PROGRAM Drain
VAR
	nSource: INT;
	nStartTimeInSeconds: UDINT ;
	nTime: UDINT;
	tempSecondsToAddWhilePause: INT;
	SecondsToAddWhilePause: INT;
	RemainingTime: UDINT;
	fb_FTRIG: R_TRIG;
	bStartCommand: BOOL;
	CLK: INT;
	Q: INT;
	b: BOOL;
	bN2PurgeBlockEnded: BOOL;
	fbSelection : FBSelection;
	

END_VAR

VAR_INPUT
	nCurrentBlock: INT;
	sSourceName: STRING;
END_VAR

fbSelection.TargetConverter(sTargetName:= sSourceName, TargetConverter_output => nSource); 


IF (RecipeTags.bStartTimeEnable[nCurrentBlock]=FALSE) THEN
	RecipeTags.Recipe.Blocks[nCurrentBlock].Properties.sStartTime:=MAIN.sConcatenatedHourMinuteString;
	nStartTimeInSeconds := STRING_TO_UDINT(MAIN.sCurrentSecond);
	RecipeTags.bStartTimeEnable[nCurrentBlock] :=  TRUE;
END_IF



IF RecipeTags.Recipe.Blocks[nCurrentBlock].Properties.sIntervalType = 'S' THEN
	nTime := DINT_TO_UDINT(RecipeTags.Recipe.Blocks[nCurrentBlock].Properties.nInterval);
ELSIF RecipeTags.Recipe.Blocks[nCurrentBlock].Properties.sIntervalType = 'M' THEN
	nTime := DINT_TO_UDINT(RecipeTags.Recipe.Blocks[nCurrentBlock].Properties.nInterval * 60);
ELSIF RecipeTags.Recipe.Blocks[nCurrentBlock].Properties.sIntervalType = 'H' THEN
	nTime := DINT_TO_UDINT(RecipeTags.Recipe.Blocks[nCurrentBlock].Properties.nInterval * 3600);
END_IF


IF RecipeTags.enWaitPause[nCurrentBlock] THEN
	tempSecondsToAddWhilePause := tempSecondsToAddWhilePause + 1;
	SecondsToAddWhilePause := tempSecondsToAddWhilePause; 
ELSE
	tempSecondsToAddWhilePause := 0;
END_IF

IF NOT(RecipeTags.bPauseRecipe) THEN
		RecipeTags.enWaitPause[nCurrentBlock] := FALSE;
		RecipeTags.bBlockStart[nCurrentBlock] := TRUE;
		RemainingTime := nTime- nStartTimeInSeconds-STRING_TO_UDINT(MAIN.sCurrentSecond);
ELSE
		RecipeTags.bBlockStart[nCurrentBlock] := FALSE;
		RecipeTags.enWaitPause[nCurrentBlock] := TRUE;
END_IF

IF  (nTime + nStartTimeInSeconds + DINT_TO_UDINT(TRUNC(SecondsToAddWhilePause/100))) <= (STRING_TO_UDINT(MAIN.sCurrentSecond)) AND RecipeTags.bSkipDrain THEN
	RecipeTags.Recipe.Blocks[nCurrentBlock].Properties.bStopCommand := TRUE;
	RecipeTags.Recipe.Blocks[nCurrentBlock].Properties.sEndTime:=MAIN.sConcatenatedHourMinuteString;
	RecipeTags.bBlockStart[nCurrentBlock] := FALSE;
	RecipeTags.bBlockEnd[nCurrentBlock] := TRUE;
	RecipeTags.bDrainStatus := FALSE;
	RecipeTags.bSkipDrain := FALSE;

ELSIF RecipeTags.bSkipDrain THEN
	RecipeTags.Recipe.Blocks[nCurrentBlock].Properties.bStopCommand := TRUE;
	RecipeTags.Recipe.Blocks[nCurrentBlock].Properties.sEndTime:=MAIN.sConcatenatedHourMinuteString;
	RecipeTags.bBlockStart[nCurrentBlock] := FALSE;
	RecipeTags.bBlockEnd[nCurrentBlock] := TRUE;
	RecipeTags.bDrainStatus := FALSE;
	RecipeTags.bSkipDrain := FALSE;
ELSE
	RecipeTags.bBlockEnd[nCurrentBlock] := FALSE;
END_IF

IF RecipeTags.bBlockStart[nCurrentBlock] THEN
	RecipeTags.bDrainStatus := TRUE;
	IF (nSource>=0 AND nSource<5) OR (nSource>6 AND nSource<=8) THEN
		IO.Vessels[nSource].Valves[0].bStart := TRUE;
	END_IF
	IF nSource=5 OR nSource=6 THEN
		IO.Vessels[nSource].Valves[6].bStart := TRUE;
		IO.Vessels[nSource].Valves[0].bStart := TRUE;
	END_IF
	//MVA drain
	IF nSource=9 AND nSource<10 THEN
		IO.Reactors[nSource-9].Valves[5].bStart := TRUE;
		IO.Reactors[nSource-9].Valves[0].bStart := TRUE;
		IO.Reactors[nSource-9].Valves[2].bStart := TRUE;
	END_IF
	//RV Drain
	IF nSource=10 OR nSource=11 THEN
		IO.Reactors[nSource-9].Valves[2].bStart := TRUE;
		IO.Reactors[nSource-9].Valves[0].bStart := TRUE;

	END_IF
ELSE
	IF (nSource>=0 AND nSource<5) OR (nSource>6 AND nSource<=8) THEN
		IO.Vessels[nSource].Valves[0].bStart := FALSE;
	END_IF
	IF nSource<9 THEN
		IO.Vessels[nSource].Valves[6].bStart := FALSE;
		IO.Vessels[nSource].Valves[0].bStart := false;

	END_IF
	//MVA drain
	IF nSource=9 AND nSource<10 THEN
		IO.Reactors[nSource-9].Valves[5].bStart := FALSE;
		IO.Reactors[nSource-9].Valves[0].bStart := FALSE;
		IO.Reactors[nSource-9].Valves[2].bStart := FALSE;
	END_IF
	IF nSource=10 OR nSource=11 THEN
		IO.Reactors[nSource-9].Valves[2].bStart := FALSE;
		IO.Reactors[nSource-9].Valves[0].bStart := FALSE;

	END_IF
END_IF

fb_FTRIG(CLK:=RecipeTags.bBlockEnd[nCurrentBlock], Q=> );
IF fb_FTRIG.Q AND RecipeTags.Recipe.Blocks[nCurrentBlock].Name = 'Drain' THEN
	RecipeTags.bSkipDrain := FALSE;
	RecipeTags.bDrainStatus := FALSE;
	RecipeTags.bBlockEnd[nCurrentBlock] := FALSE;
	RecipeTags.bStartTimeEnable[nCurrentBlock] :=  FALSE;
	SecondsToAddWhilePause := 0;
	nTime := 0;
	nStartTimeInSeconds := 0;
	RecipeTags.Recipe.Blocks[nCurrentBlock].Properties.sEndTime:=MAIN.sConcatenatedHourMinuteString;
	RecipeTags.Recipe.Blocks[nCurrentBlock].Properties.bStopCommand := TRUE;
END_IF

END_PROGRAM

(* stored: Version 1.1.0.1, ProductVersion 3.1.4024.5
   POU Drain: Id {732252c0-8d85-472e-b5c9-8a1b06f29836}, SpecialFunc None *)
